FUNCTION_BLOCK FB_Measuring
VAR_INPUT
	VIn		:	REAL;
END_VAR
VAR_OUTPUT
	EndMeasure	:	BOOL;
	
END_VAR
VAR_IN_OUT
	VOut		:	REAL;
END_VAR
VAR
	VPrev	:	REAL	:=	10.0;
	fbTonEndMeasure	:	TON;
	En : BOOL;
END_VAR

IF VIn < VPrev OR VIn > 7.3 THEN
    VPrev := VIn;
    En := VIn < VPrev; (* En sarà TRUE solo se VIn < VPrev *)
END_IF

IF En THEN
    Vout := VPrev;
END_IF

END_FUNCTION_BLOCK

(* stored: Version 1.1.0.1, ProductVersion 3.1.4024.12
   POU FB_Measuring: Id {034a35b7-d330-49e5-930f-261d0624b988}, SpecialFunc None *)
